{attribute 'qualified_only'}
VAR_GLOBAL
	fCylValveOut : REAL;
	fWinchValveOut : REAL; 
	bGreenLight : BOOL;
	bRedLight : BOOL; 
	bEnableWinchValve : BOOL;
	bEnableCylValve : BOOL; 	
END_VAR

(* stored: Version 1.1.0.1, ProductVersion 3.1.4024.12
   GVL G_Outputs: Id {b5d6af70-061f-45ef-b52a-5693aeee88d7} *)
